# EPICS substitutions: TPGSup/TPG300_switching_functions.substitutions
file TPG300_switching_functions.template {

pattern {PORT, P, Q}
{"\$(PORT)", "\$(P)", "SEL"}
{"\$(PORT)", "\$(P)", "1"}
{"\$(PORT)", "\$(P)", "2"}
{"\$(PORT)", "\$(P)", "3"}
{"\$(PORT)", "\$(P)", "4"}
{"\$(PORT)", "\$(P)", "A"}
{"\$(PORT)", "\$(P)", "B"}

}
